SPLINE
SPL {X  -162.485, Y  +370.062, Z    +0.000, E1   +10.606, E3 +598080.502}
SPL {X  -162.818, Y  +379.636, Z    +0.000, E1    +5.115, E3 +598069.851}
SPL {X  -162.820, Y  +386.976, Z    +0.000, E1    +0.144, E3 +598068.950}
SPL {X  -162.820, Y  +391.982, Z    +0.000, E1    -3.443, E3 +598075.715}
SPL {X  -162.820, Y  +399.630, Z    +0.000, E1    -9.426, E3 +598078.222}
SPL {X  -162.820, Y  +408.127, Z    +0.000, E1   -18.417, E3 +598064.510}
SPL {X  -162.820, Y  +420.083, Z    +0.000, E1   -24.325, E3 +598084.986}
SPL {X  -162.820, Y  +428.527, Z    +0.000, E1   -26.988, E3 +598102.278}
SPL {X  -162.820, Y  +431.191, Z    +0.000, E1   -23.548, E3 +598137.131}
SPL {X  -162.820, Y  +432.946, Z    +0.000, E1   -22.795, E3 +598151.534}
SPL {X  -162.820, Y  +434.888, Z    +0.000, E1   -22.823, E3 +598160.941}
SPL {X  -162.820, Y  +436.834, Z    +0.000, E1   -22.779, E3 +598170.901}
SPL {X  -162.820, Y  +438.868, Z    +0.000, E1   -22.837, E3 +598180.555}
SPL {X  -162.820, Y  +441.351, Z    +0.000, E1   -22.805, E3 +598193.130}
SPL {X  -162.820, Y  +443.809, Z    +0.000, E1   -22.804, E3 +598205.296}
SPL {X  -162.820, Y  +446.105, Z    +0.000, E1   -22.815, E3 +598216.539}
SPL {X  -162.820, Y  +447.974, Z    +0.000, E1   -22.856, E3 +598225.441}
SPL {X  -162.820, Y  +449.911, Z    +0.000, E1   -22.774, E3 +598235.716}
SPL {X  -162.820, Y  +451.861, Z    +0.000, E1   -22.750, E3 +598245.564}
SPL {X  -162.820, Y  +454.167, Z    +0.000, E1   -22.842, E3 +598256.293}
SPL {X  -162.820, Y  +456.529, Z    +0.000, E1   -22.855, E3 +598267.822}
SPL {X  -162.820, Y  +458.725, Z    +0.000, E1   -22.793, E3 +598279.226}
SPL {X  -162.820, Y  +461.700, Z    +0.000, E1   -22.822, E3 +598293.849}
SPL {X  -162.820, Y  +464.633, Z    +0.000, E1   -22.813, E3 +598308.345}
SPL {X  -162.820, Y  +466.699, Z    +0.000, E1   -22.824, E3 +598318.391}
SPL {X  -162.820, Y  +468.655, Z    +0.000, E1   -22.858, E3 +598327.835}
SPL {X  -162.820, Y  +470.892, Z    +0.000, E1   -22.837, E3 +598339.074}
SPL {X  -162.820, Y  +473.485, Z    +0.000, E1   -22.806, E3 +598352.272}
SPL {X  -162.820, Y  +475.738, Z    +0.000, E1   -22.728, E3 +598363.937}
SPL {X  -162.820, Y  +478.177, Z    +0.000, E1   -22.834, E3 +598375.277}
SPL {X  -162.820, Y  +481.034, Z    +0.000, E1   -22.831, E3 +598389.414}
SPL {X  -162.820, Y  +483.391, Z    +0.000, E1   -22.793, E3 +598401.350}
SPL {X  -162.820, Y  +486.307, Z    +0.000, E1   -22.833, E3 +598415.604}
SPL {X  -162.820, Y  +489.750, Z    +0.000, E1   -22.832, E3 +598432.674}
SPL {X  -162.820, Y  +493.233, Z    +0.000, E1   -22.844, E3 +598449.811}
SPL {X  -162.820, Y  +496.150, Z    +0.000, E1   -22.796, E3 +598464.531}
SPL {X  -162.820, Y  +498.661, Z    +0.000, E1   -22.828, E3 +598476.712}
SPL {X  -162.820, Y  +501.761, Z    +0.000, E1   -22.820, E3 +598492.280}
SPL {X  -162.820, Y  +505.323, Z    +0.000, E1   -22.838, E3 +598509.727}
SPL {X  -162.820, Y  +507.875, Z    +0.000, E1   -22.849, E3 +598522.094}
SPL {X  -162.820, Y  +510.068, Z    +0.000, E1   -22.761, E3 +598533.787}
SPL {X  -162.820, Y  +512.359, Z    +0.000, E1   -22.823, E3 +598544.519}
SPL {X  -162.820, Y  +514.562, Z    +0.000, E1   -22.806, E3 +598555.706}
SPL {X  -162.820, Y  +517.952, Z    +0.000, E1   -22.864, E3 +598572.103}
SPL {X  -162.820, Y  +520.641, Z    +0.000, E1   -22.790, E3 +598585.821}
SPL {X  -162.820, Y  +522.740, Z    +0.000, E1   -22.811, E3 +598596.064}
SPL {X  -162.820, Y  +525.255, Z    +0.000, E1   -22.822, E3 +598608.484}
SPL {X  -162.820, Y  +528.050, Z    +0.000, E1   -22.808, E3 +598622.449}
SPL {X  -162.820, Y  +530.303, Z    +0.000, E1   -22.798, E3 +598633.603}
SPL {X  -162.820, Y  +532.614, Z    +0.000, E1   -22.828, E3 +598644.871}
SPL {X  -162.820, Y  +534.838, Z    +0.000, E1   -22.864, E3 +598655.500}
SPL {X  -162.820, Y  +536.882, Z    +0.000, E1   -22.782, E3 +598666.355}
SPL {X  -162.820, Y  +539.194, Z    +0.000, E1   -22.826, E3 +598677.404}
SPL {X  -162.820, Y  +541.555, Z    +0.000, E1   -22.817, E3 +598689.218}
SPL {X  -162.820, Y  +543.728, Z    +0.000, E1   -22.799, E3 +598700.076}
SPL {X  -162.820, Y  +545.925, Z    +0.000, E1   -22.803, E3 +598710.945}
SPL {X  -162.820, Y  +548.328, Z    +0.000, E1   -22.796, E3 +598722.941}
SPL {X  -162.820, Y  +551.027, Z    +0.000, E1   -22.819, E3 +598736.134}
SPL {X  -162.820, Y  +553.721, Z    +0.000, E1   -22.807, E3 +598749.578}
SPL {X  -162.820, Y  +556.430, Z    +0.000, E1   -22.821, E3 +598762.874}
SPL {X  -162.820, Y  +559.675, Z    +0.000, E1   -22.837, E3 +598778.954}
SPL {X  -162.820, Y  +562.799, Z    +0.000, E1   -22.814, E3 +598794.460}
SPL {X  -162.820, Y  +565.170, Z    +0.000, E1   -22.801, E3 +598806.285}
SPL {X  -162.820, Y  +568.020, Z    +0.000, E1   -22.787, E3 +598820.672}
SPL {X  -162.820, Y  +570.992, Z    +0.000, E1   -22.834, E3 +598834.891}
SPL {X  -162.820, Y  +573.634, Z    +0.000, E1   -22.827, E3 +598848.069}
SPL {X  -162.820, Y  +576.228, Z    +0.000, E1   -22.814, E3 +598860.965}
SPL {X  -162.820, Y  +578.553, Z    +0.000, E1   -22.801, E3 +598872.581}
SPL {X  -162.820, Y  +581.064, Z    +0.000, E1   -22.823, E3 +598884.866}
SPL {X  -162.820, Y  +583.435, Z    +0.000, E1   -22.808, E3 +598896.687}
SPL {X  -162.820, Y  +585.410, Z    +0.000, E1   -22.764, E3 +598906.823}
SPL {X  -162.820, Y  +587.676, Z    +0.000, E1   -22.853, E3 +598917.338}
SPL {X  -162.820, Y  +589.682, Z    +0.000, E1   -22.776, E3 +598927.868}
SPL {X  -162.820, Y  +591.720, Z    +0.000, E1   -22.868, E3 +598937.178}
SPL {X  -162.820, Y  +593.650, Z    +0.000, E1   -22.810, E3 +598947.248}
SPL {X  -162.820, Y  +595.830, Z    +0.000, E1   -22.828, E3 +598957.864}
SPL {X  -162.820, Y  +598.094, Z    +0.000, E1   -22.843, E3 +598968.977}
SPL {X  -162.820, Y  +600.420, Z    +0.000, E1   -22.826, E3 +598980.608}
SPL {X  -162.820, Y  +602.573, Z    +0.000, E1   -22.830, E3 +598991.194}
SPL {X  -162.820, Y  +604.828, Z    +0.000, E1   -22.784, E3 +599002.832}
SPL {X  -162.820, Y  +608.133, Z    +0.000, E1   -22.831, E3 +599018.950}
SPL {X  -162.820, Y  +611.103, Z    +0.000, E1   -22.785, E3 +599033.876}
SPL {X  -162.820, Y  +613.294, Z    +0.000, E1   -22.780, E3 +599044.749}
SPL {X  -162.820, Y  +615.356, Z    +0.000, E1   -22.799, E3 +599054.806}
SPL {X  -162.820, Y  +617.439, Z    +0.000, E1   -22.808, E3 +599065.064}
SPL {X  -162.820, Y  +619.665, Z    +0.000, E1   -22.817, E3 +599076.032}
SPL {X  -162.820, Y  +621.733, Z    +0.000, E1   -22.759, E3 +599086.756}
SPL {X  -162.820, Y  +624.076, Z    +0.000, E1   -22.774, E3 +599098.261}
SPL {X  -162.820, Y  +626.527, Z    +0.000, E1   -22.768, E3 +599110.504}
SPL {X  -162.820, Y  +629.758, Z    +0.000, E1   -22.800, E3 +599126.433}
SPL {X  -162.820, Y  +632.572, Z    +0.000, E1   -22.785, E3 +599140.282}
SPL {X  -162.820, Y  +634.507, Z    +0.000, E1   -22.784, E3 +599149.921}
SPL {X  -162.820, Y  +636.863, Z    +0.000, E1   -22.760, E3 +599161.843}
SPL {X  -162.820, Y  +640.111, Z    +0.000, E1   -22.809, E3 +599177.726}
SPL {X  -162.820, Y  +643.449, Z    +0.000, E1   -22.796, E3 +599194.244}
SPL {X  -162.820, Y  +645.630, Z    +0.000, E1   -22.795, E3 +599204.940}
SPL {X  -162.820, Y  +647.561, Z    +0.000, E1   -22.705, E3 +599215.390}
SPL {X  -162.820, Y  +649.758, Z    +0.000, E1   -22.780, E3 +599225.581}
SPL {X  -162.820, Y  +651.708, Z    +0.000, E1   -22.810, E3 +599235.075}
SPL {X  -162.820, Y  +653.898, Z    +0.000, E1   -22.796, E3 +599245.996}
SPL {X  -162.820, Y  +656.161, Z    +0.000, E1   -22.812, E3 +599257.117}
SPL {X  -162.820, Y  +658.384, Z    +0.000, E1   -22.822, E3 +599267.983}
SPL {X  -162.820, Y  +660.215, Z    +0.000, E1   -22.649, E3 +599278.574}
SPL {X  -162.820, Y  +662.823, Z    +0.000, E1   -22.799, E3 +599290.282}
SPL {X  -162.820, Y  +665.112, Z    +0.000, E1   -22.835, E3 +599301.336}
SPL {X  -162.820, Y  +667.016, Z    +0.000, E1   -22.823, E3 +599310.765}
SPL {X  -162.820, Y  +668.960, Z    +0.000, E1   -22.773, E3 +599320.932}
SPL {X  -162.820, Y  +672.333, Z    +0.000, E1   -22.837, E3 +599337.268}
SPL {X  -162.812, Y  +675.071, Z    +0.000, E1   -22.742, E3 +599351.413}
SPL {X  -162.773, Y  +677.428, Z    +0.000, E1   -22.762, E3 +599363.011}
SPL {X  -162.691, Y  +679.987, Z    +0.000, E1   -22.794, E3 +599375.424}
SPL {X  -162.604, Y  +681.880, Z    +0.000, E1   -22.691, E3 +599385.585}
SPL {X  -162.458, Y  +684.346, Z    +0.000, E1   -22.764, E3 +599397.379}
SPL {X  -162.296, Y  +686.547, Z    +0.000, E1   -22.660, E3 +599408.996}
SPL {X  -162.164, Y  +688.106, Z    +0.000, E1   -22.661, E3 +599416.729}
SPL {X  -161.938, Y  +690.422, Z    +0.000, E1   -22.769, E3 +599427.405}
SPL {X  -161.065, Y  +697.344, Z    +0.000, E1   -25.698, E3 +599436.524}
SPL {X  -158.730, Y  +709.763, Z    +0.000, E1   -31.225, E3 +599445.197}
ENDSPLINE

SPLINE
SPL {X  -160.932, Y  +698.225, Z    +0.000, E1   -21.712, E3 +599476.307}
SPL {X  -161.917, Y  +690.622, Z    +0.000, E1   -16.445, E3 +599489.907}
ENDSPLINE

SPLINE
SPL {X  -161.349, Y  +695.340, Z    +0.000, E1   -18.625, E3 +599497.526}
ENDSPLINE

SPLINE
SPL {X  -162.534, Y  +683.153, Z    +0.000, E1   -10.475, E3 +599518.657}
SPL {X  -162.820, Y  +667.630, Z    +0.000, E1    -0.882, E3 +599512.633}
SPL {X  -162.820, Y  +661.883, Z    +0.000, E1    +3.373, E3 +599518.076}
SPL {X  -162.820, Y  +655.163, Z    +0.000, E1    +8.702, E3 +599517.675}
SPL {X  -162.820, Y  +634.515, Z    +0.000, E1   +26.439, E3 +599510.088}
ENDSPLINE

SPLINE
SPL {X  -162.820, Y  +638.080, Z    +0.000, E1   +18.858, E3 +599540.053}
ENDSPLINE

SPLINE
SPL {X  -162.820, Y  +623.278, Z    +0.000, E1   +28.723, E3 +599541.623}
SPL {X  -162.820, Y  +618.658, Z    +0.000, E1   +26.841, E3 +599570.232}
ENDSPLINE

SPLINE
SPL {X  -162.820, Y  +623.685, Z    +0.000, E1   +22.346, E3 +599582.539}
ENDSPLINE

SPLINE
SPL {X  -162.820, Y  +621.304, Z    +0.000, E1   +22.259, E3 +599595.354}
SPL {X  -162.820, Y  +618.758, Z    +0.000, E1   +22.239, E3 +599608.505}
SPL {X  -162.820, Y  +616.062, Z    +0.000, E1   +22.275, E3 +599621.925}
SPL {X  -162.820, Y  +613.536, Z    +0.000, E1   +22.242, E3 +599635.047}
SPL {X  -162.820, Y  +610.461, Z    +0.000, E1   +22.264, E3 +599650.678}
SPL {X  -162.820, Y  +607.796, Z    +0.000, E1   +22.261, E3 +599664.049}
SPL {X  -162.820, Y  +605.178, Z    +0.000, E1   +22.267, E3 +599677.533}
SPL {X  -162.820, Y  +602.350, Z    +0.000, E1   +22.224, E3 +599692.150}
SPL {X  -162.820, Y  +599.842, Z    +0.000, E1   +22.298, E3 +599704.302}
SPL {X  -162.820, Y  +597.194, Z    +0.000, E1   +22.253, E3 +599718.223}
SPL {X  -162.820, Y  +594.115, Z    +0.000, E1   +22.273, E3 +599733.752}
SPL {X  -162.820, Y  +591.721, Z    +0.000, E1   +22.239, E3 +599746.067}
SPL {X  -162.820, Y  +589.492, Z    +0.000, E1   +22.304, E3 +599756.928}
SPL {X  -162.820, Y  +587.447, Z    +0.000, E1   +22.279, E3 +599767.457}
SPL {X  -162.820, Y  +585.192, Z    +0.000, E1   +22.298, E3 +599778.867}
SPL {X  -162.820, Y  +582.610, Z    +0.000, E1   +22.234, E3 +599792.490}
SPL {X  -162.820, Y  +580.317, Z    +0.000, E1   +22.300, E3 +599803.544}
SPL {X  -162.820, Y  +578.878, Z    +0.000, E1   +22.272, E3 +599811.054}
SPL {X  -162.820, Y  +576.856, Z    +0.000, E1   +22.233, E3 +599821.812}
SPL {X  -162.820, Y  +574.811, Z    +0.000, E1   +22.236, E3 +599832.076}
SPL {X  -162.820, Y  +572.645, Z    +0.000, E1   +22.246, E3 +599843.171}
SPL {X  -162.820, Y  +569.475, Z    +0.000, E1   +22.269, E3 +599859.177}
SPL {X  -162.820, Y  +565.838, Z    +0.000, E1   +22.271, E3 +599877.772}
SPL {X  -162.820, Y  +562.162, Z    +0.000, E1   +22.252, E3 +599896.589}
SPL {X  -162.820, Y  +559.515, Z    +0.000, E1   +22.273, E3 +599909.708}
SPL {X  -162.820, Y  +556.723, Z    +0.000, E1   +22.309, E3 +599923.792}
SPL {X  -162.820, Y  +553.294, Z    +0.000, E1   +22.266, E3 +599941.579}
SPL {X  -162.820, Y  +550.136, Z    +0.000, E1   +22.258, E3 +599957.693}
SPL {X  -162.820, Y  +546.694, Z    +0.000, E1   +22.290, E3 +599975.015}
SPL {X  -162.820, Y  +543.558, Z    +0.000, E1   +22.285, E3 +599990.878}
SPL {X  -162.820, Y  +541.633, Z    +0.000, E1   +22.257, E3 +600000.806}
SPL {X  -162.820, Y  +539.116, Z    +0.000, E1   +22.302, E3 +600013.416}
SPL {X  -162.820, Y  +536.913, Z    +0.000, E1   +22.192, E3 +600025.341}
SPL {X  -162.820, Y  +534.880, Z    +0.000, E1   +22.252, E3 +600035.294}
SPL {X  -162.820, Y  +532.896, Z    +0.000, E1   +22.234, E3 +600045.455}
SPL {X  -162.820, Y  +531.056, Z    +0.000, E1   +22.251, E3 +600054.737}
SPL {X  -162.820, Y  +528.708, Z    +0.000, E1   +22.319, E3 +600066.118}
SPL {X  -162.820, Y  +525.932, Z    +0.000, E1   +22.258, E3 +600080.875}
SPL {X  -162.820, Y  +522.524, Z    +0.000, E1   +22.326, E3 +600097.598}
SPL {X  -162.820, Y  +519.457, Z    +0.000, E1   +22.481, E3 +600111.727}
SPL {X  -162.820, Y  +506.285, Z    +0.000, E1   +28.538, E3 +600123.185}
SPL {X  -162.820, Y  +504.441, Z    +0.000, E1   +27.574, E3 +600137.528}
SPL {X  -162.820, Y  +502.813, Z    +0.000, E1   +26.013, E3 +600155.725}
SPL {X  -162.820, Y  +502.016, Z    +0.000, E1   +24.802, E3 +600168.068}
SPL {X  -162.820, Y  +501.060, Z    +0.000, E1   +24.081, E3 +600178.257}
SPL {X  -162.820, Y  +499.934, Z    +0.000, E1   +22.814, E3 +600194.126}
SPL {X  -162.820, Y  +498.303, Z    +0.000, E1   +21.749, E3 +600211.382}
SPL {X  -162.820, Y  +495.897, Z    +0.000, E1   +21.662, E3 +600224.536}
SPL {X  -162.820, Y  +493.717, Z    +0.000, E1   +21.704, E3 +600235.642}
SPL {X  -162.820, Y  +491.396, Z    +0.000, E1   +21.707, E3 +600247.766}
SPL {X  -162.820, Y  +489.485, Z    +0.000, E1   +21.661, E3 +600258.114}
SPL {X  -162.820, Y  +487.723, Z    +0.000, E1   +21.665, E3 +600267.317}
SPL {X  -162.820, Y  +485.661, Z    +0.000, E1   +21.712, E3 +600277.761}
SPL {X  -162.820, Y  +482.775, Z    +0.000, E1   +21.716, E3 +600293.013}
SPL {X  -162.820, Y  +479.894, Z    +0.000, E1   +21.695, E3 +600308.089}
SPL {X  -162.820, Y  +477.685, Z    +0.000, E1   +21.656, E3 +600320.027}
SPL {X  -162.820, Y  +475.419, Z    +0.000, E1   +21.711, E3 +600331.380}
SPL {X  -162.820, Y  +473.301, Z    +0.000, E1   +21.712, E3 +600342.477}
SPL {X  -162.820, Y  +470.965, Z    +0.000, E1   +21.700, E3 +600354.822}
SPL {X  -162.820, Y  +469.036, Z    +0.000, E1   +21.695, E3 +600364.865}
SPL {X  -162.820, Y  +467.138, Z    +0.000, E1   +21.678, E3 +600375.037}
SPL {X  -162.820, Y  +465.011, Z    +0.000, E1   +21.692, E3 +600386.020}
SPL {X  -162.820, Y  +462.669, Z    +0.000, E1   +21.752, E3 +600397.800}
SPL {X  -162.820, Y  +460.725, Z    +0.000, E1   +21.689, E3 +600408.413}
SPL {X  -162.820, Y  +458.666, Z    +0.000, E1   +21.695, E3 +600419.225}
SPL {X  -162.820, Y  +456.431, Z    +0.000, E1   +21.708, E3 +600430.753}
SPL {X  -162.820, Y  +454.628, Z    +0.000, E1   +21.674, E3 +600440.472}
SPL {X  -162.820, Y  +452.690, Z    +0.000, E1   +21.773, E3 +600449.746}
SPL {X  -162.820, Y  +450.610, Z    +0.000, E1   +21.698, E3 +600461.345}
SPL {X  -162.820, Y  +448.170, Z    +0.000, E1   +21.667, E3 +600474.365}
SPL {X  -162.820, Y  +446.246, Z    +0.000, E1   +21.696, E3 +600484.183}
SPL {X  -162.820, Y  +443.784, Z    +0.000, E1   +21.713, E3 +600496.969}
SPL {X  -162.820, Y  +440.567, Z    +0.000, E1   +21.731, E3 +600513.809}
SPL {X  -162.820, Y  +437.628, Z    +0.000, E1   +21.678, E3 +600529.473}
SPL {X  -162.820, Y  +435.262, Z    +0.000, E1   +21.727, E3 +600541.409}
SPL {X  -162.820, Y  +433.510, Z    +0.000, E1   +21.692, E3 +600550.823}
SPL {X  -162.820, Y  +431.492, Z    +0.000, E1   +21.686, E3 +600561.518}
SPL {X  -162.820, Y  +429.074, Z    +0.000, E1   +21.710, E3 +600573.970}
SPL {X  -162.820, Y  +427.020, Z    +0.000, E1   +21.674, E3 +600584.972}
SPL {X  -162.820, Y  +424.525, Z    +0.000, E1   +21.712, E3 +600597.885}
SPL {X  -162.820, Y  +421.144, Z    +0.000, E1   +21.719, E3 +600615.552}
SPL {X  -162.820, Y  +418.116, Z    +0.000, E1   +21.761, E3 +600630.883}
SPL {X  -162.820, Y  +416.127, Z    +0.000, E1   +21.715, E3 +600641.588}
SPL {X  -162.820, Y  +414.361, Z    +0.000, E1   +21.613, E3 +600651.775}
SPL {X  -162.820, Y  +412.134, Z    +0.000, E1   +21.697, E3 +600662.720}
SPL {X  -162.820, Y  +409.248, Z    +0.000, E1   +21.741, E3 +600677.655}
SPL {X  -162.820, Y  +406.238, Z    +0.000, E1   +21.697, E3 +600693.623}
SPL {X  -162.820, Y  +404.001, Z    +0.000, E1   +21.723, E3 +600705.053}
SPL {X  -162.820, Y  +402.223, Z    +0.000, E1   +21.697, E3 +600714.538}
SPL {X  -162.820, Y  +400.348, Z    +0.000, E1   +21.713, E3 +600724.264}
SPL {X  -162.820, Y  +398.298, Z    +0.000, E1   +21.721, E3 +600734.879}
SPL {X  -162.820, Y  +396.371, Z    +0.000, E1   +21.713, E3 +600745.061}
SPL {X  -162.820, Y  +394.508, Z    +0.000, E1   +21.616, E3 +600755.617}
SPL {X  -162.820, Y  +392.435, Z    +0.000, E1   +21.681, E3 +600765.970}
SPL {X  -162.820, Y  +389.390, Z    +0.000, E1   +21.742, E3 +600781.577}
SPL {X  -162.820, Y  +386.818, Z    +0.000, E1   +21.679, E3 +600795.336}
SPL {X  -162.820, Y  +384.697, Z    +0.000, E1   +21.693, E3 +600806.406}
SPL {X  -162.820, Y  +382.288, Z    +0.000, E1   +21.742, E3 +600818.529}
SPL {X  -162.817, Y  +379.520, Z    +0.000, E1   +21.723, E3 +600833.367}
SPL {X  -162.776, Y  +376.710, Z    +0.000, E1   +21.698, E3 +600848.106}
SPL {X  -162.707, Y  +374.438, Z    +0.000, E1   +21.688, E3 +600860.110}
SPL {X  -162.607, Y  +372.171, Z    +0.000, E1   +21.692, E3 +600871.910}
SPL {X  -162.494, Y  +370.197, Z    +0.000, E1   +21.655, E3 +600882.536}
SPL {X  -162.349, Y  +368.131, Z    +0.000, E1   +21.624, E3 +600893.654}
SPL {X  -162.161, Y  +365.866, Z    +0.000, E1   +21.642, E3 +600905.339}
SPL {X  -161.651, Y  +361.024, Z    +0.000, E1   +22.970, E3 +600918.762}
SPL {X  -160.281, Y  +351.857, Z    +0.000, E1   +24.243, E3 +600954.101}
ENDSPLINE

SPLINE
SPL {X  -161.833, Y  +362.603, Z    +0.000, E1   +17.021, E3 +600968.797}
ENDSPLINE

SPLINE
SPL {X  -160.786, Y  +354.842, Z    +0.000, E1   +19.274, E3 +601000.953}
ENDSPLINE

SPLINE
SPL {X  -162.485, Y  +370.062, Z    +0.000, E1   +10.606, E3 +601007.331}
SPL {X  -162.818, Y  +379.636, Z    +0.000, E1    +5.115, E3 +600996.680}
SPL {X  -162.820, Y  +386.976, Z    +0.000, E1    +0.144, E3 +600995.779}
SPL {X  -162.820, Y  +391.982, Z    +0.000, E1    -3.443, E3 +601002.544}
SPL {X  -162.820, Y  +399.630, Z    +0.000, E1    -9.426, E3 +601005.051}
SPL {X  -162.820, Y  +408.127, Z    +0.000, E1   -18.417, E3 +600991.340}
SPL {X  -162.820, Y  +420.083, Z    +0.000, E1   -24.325, E3 +601011.815}
SPL {X  -162.820, Y  +428.527, Z    +0.000, E1   -26.988, E3 +601029.107}
SPL {X  -162.820, Y  +431.336, Z    +0.000, E1   -24.162, E3 +601059.317}
SPL {X  -162.820, Y  +432.048, Z    +0.000, E1   -22.832, E3 +601073.821}
SPL {X  -162.820, Y  +434.888, Z    +0.000, E1   -22.823, E3 +601087.770}
SPL {X  -162.820, Y  +436.834, Z    +0.000, E1   -22.779, E3 +601097.730}
SPL {X  -162.820, Y  +438.868, Z    +0.000, E1   -22.837, E3 +601107.384}
SPL {X  -162.820, Y  +441.351, Z    +0.000, E1   -22.805, E3 +601119.959}
SPL {X  -162.820, Y  +443.809, Z    +0.000, E1   -22.804, E3 +601132.126}
SPL {X  -162.820, Y  +446.105, Z    +0.000, E1   -22.815, E3 +601143.368}
SPL {X  -162.820, Y  +447.974, Z    +0.000, E1   -22.856, E3 +601152.271}
SPL {X  -162.820, Y  +449.911, Z    +0.000, E1   -22.774, E3 +601162.546}
SPL {X  -162.820, Y  +451.861, Z    +0.000, E1   -22.750, E3 +601172.393}
SPL {X  -162.820, Y  +454.167, Z    +0.000, E1   -22.842, E3 +601183.123}
SPL {X  -162.820, Y  +456.529, Z    +0.000, E1   -22.855, E3 +601194.651}
SPL {X  -162.820, Y  +458.725, Z    +0.000, E1   -22.793, E3 +601206.055}
SPL {X  -162.820, Y  +460.754, Z    +0.000, E1   -22.806, E3 +601215.928}
SPL {X  -162.820, Y  +462.409, Z    +0.000, E1   -22.783, E3 +601224.345}
SPL {X  -162.820, Y  +464.633, Z    +0.000, E1   -22.813, E3 +601235.175}
SPL {X  -162.820, Y  +467.913, Z    +0.000, E1   -22.879, E3 +601251.014}
SPL {X  -162.820, Y  +470.892, Z    +0.000, E1   -22.837, E3 +601265.903}
SPL {X  -162.820, Y  +472.726, Z    +0.000, E1   -22.777, E3 +601275.442}
SPL {X  -162.820, Y  +475.118, Z    +0.000, E1   -22.777, E3 +601287.413}
SPL {X  -162.820, Y  +477.389, Z    +0.000, E1   -22.803, E3 +601298.330}
SPL {X  -162.820, Y  +478.914, Z    +0.000, E1   -22.821, E3 +601305.721}
SPL {X  -162.820, Y  +481.034, Z    +0.000, E1   -22.831, E3 +601316.244}
SPL {X  -162.820, Y  +484.256, Z    +0.000, E1   -22.840, E3 +601332.262}
SPL {X  -162.820, Y  +487.952, Z    +0.000, E1   -22.824, E3 +601350.692}
SPL {X  -162.820, Y  +490.653, Z    +0.000, E1   -22.810, E3 +601363.962}
SPL {X  -162.820, Y  +493.233, Z    +0.000, E1   -22.844, E3 +601376.640}
SPL {X  -162.820, Y  +496.150, Z    +0.000, E1   -22.796, E3 +601391.360}
SPL {X  -162.820, Y  +498.661, Z    +0.000, E1   -22.828, E3 +601403.541}
SPL {X  -162.820, Y  +501.761, Z    +0.000, E1   -22.820, E3 +601419.109}
SPL {X  -162.820, Y  +505.323, Z    +0.000, E1   -22.838, E3 +601436.556}
SPL {X  -162.820, Y  +507.875, Z    +0.000, E1   -22.849, E3 +601448.923}
SPL {X  -162.820, Y  +510.068, Z    +0.000, E1   -22.761, E3 +601460.616}
SPL {X  -162.820, Y  +512.359, Z    +0.000, E1   -22.823, E3 +601471.348}
SPL {X  -162.820, Y  +514.562, Z    +0.000, E1   -22.806, E3 +601482.535}
SPL {X  -162.820, Y  +517.952, Z    +0.000, E1   -22.864, E3 +601498.932}
SPL {X  -162.820, Y  +520.641, Z    +0.000, E1   -22.790, E3 +601512.651}
SPL {X  -162.820, Y  +522.740, Z    +0.000, E1   -22.811, E3 +601522.893}
SPL {X  -162.820, Y  +524.628, Z    +0.000, E1   -22.846, E3 +601531.888}
SPL {X  -162.820, Y  +526.661, Z    +0.000, E1   -22.801, E3 +601542.444}
SPL {X  -162.820, Y  +529.662, Z    +0.000, E1   -22.810, E3 +601557.294}
SPL {X  -162.820, Y  +532.614, Z    +0.000, E1   -22.828, E3 +601571.701}
SPL {X  -162.820, Y  +534.838, Z    +0.000, E1   -22.864, E3 +601582.330}
SPL {X  -162.820, Y  +536.882, Z    +0.000, E1   -22.782, E3 +601593.184}
SPL {X  -162.820, Y  +539.194, Z    +0.000, E1   -22.826, E3 +601604.233}
SPL {X  -162.820, Y  +541.555, Z    +0.000, E1   -22.817, E3 +601616.047}
SPL {X  -162.820, Y  +543.728, Z    +0.000, E1   -22.799, E3 +601626.905}
SPL {X  -162.820, Y  +545.925, Z    +0.000, E1   -22.803, E3 +601637.775}
SPL {X  -162.820, Y  +548.328, Z    +0.000, E1   -22.796, E3 +601649.770}
SPL {X  -162.820, Y  +551.027, Z    +0.000, E1   -22.819, E3 +601662.963}
SPL {X  -162.820, Y  +553.721, Z    +0.000, E1   -22.807, E3 +601676.407}
SPL {X  -162.820, Y  +556.430, Z    +0.000, E1   -22.821, E3 +601689.703}
SPL {X  -162.820, Y  +558.974, Z    +0.000, E1   -22.806, E3 +601702.403}
SPL {X  -162.820, Y  +562.171, Z    +0.000, E1   -22.845, E3 +601718.101}
SPL {X  -162.820, Y  +565.170, Z    +0.000, E1   -22.801, E3 +601733.115}
SPL {X  -162.820, Y  +567.308, Z    +0.000, E1   -22.750, E3 +601744.131}
SPL {X  -162.820, Y  +570.378, Z    +0.000, E1   -22.843, E3 +601758.755}
SPL {X  -162.820, Y  +573.634, Z    +0.000, E1   -22.827, E3 +601774.898}
SPL {X  -162.820, Y  +576.228, Z    +0.000, E1   -22.814, E3 +601787.795}
SPL {X  -162.820, Y  +578.553, Z    +0.000, E1   -22.801, E3 +601799.411}
SPL {X  -162.820, Y  +581.064, Z    +0.000, E1   -22.823, E3 +601811.695}
SPL {X  -162.820, Y  +583.435, Z    +0.000, E1   -22.808, E3 +601823.517}
SPL {X  -162.820, Y  +585.410, Z    +0.000, E1   -22.764, E3 +601833.652}
SPL {X  -162.820, Y  +587.676, Z    +0.000, E1   -22.853, E3 +601844.167}
SPL {X  -162.820, Y  +590.707, Z    +0.000, E1   -22.855, E3 +601859.317}
SPL {X  -162.820, Y  +593.650, Z    +0.000, E1   -22.810, E3 +601874.078}
SPL {X  -162.820, Y  +595.830, Z    +0.000, E1   -22.828, E3 +601884.693}
SPL {X  -162.820, Y  +598.094, Z    +0.000, E1   -22.843, E3 +601895.807}
SPL {X  -162.820, Y  +600.420, Z    +0.000, E1   -22.826, E3 +601907.438}
SPL {X  -162.820, Y  +602.573, Z    +0.000, E1   -22.830, E3 +601918.023}
SPL {X  -162.820, Y  +604.828, Z    +0.000, E1   -22.784, E3 +601929.661}
SPL {X  -162.820, Y  +608.133, Z    +0.000, E1   -22.831, E3 +601945.779}
SPL {X  -162.820, Y  +611.103, Z    +0.000, E1   -22.785, E3 +601960.705}
SPL {X  -162.820, Y  +613.294, Z    +0.000, E1   -22.780, E3 +601971.578}
SPL {X  -162.820, Y  +615.356, Z    +0.000, E1   -22.799, E3 +601981.635}
SPL {X  -162.820, Y  +617.439, Z    +0.000, E1   -22.808, E3 +601991.893}
SPL {X  -162.820, Y  +619.665, Z    +0.000, E1   -22.817, E3 +602002.861}
SPL {X  -162.820, Y  +621.733, Z    +0.000, E1   -22.759, E3 +602013.586}
SPL {X  -162.820, Y  +624.076, Z    +0.000, E1   -22.774, E3 +602025.091}
SPL {X  -162.820, Y  +627.244, Z    +0.000, E1   -22.803, E3 +602040.773}
SPL {X  -162.820, Y  +630.349, Z    +0.000, E1   -22.766, E3 +602056.305}
SPL {X  -162.820, Y  +632.572, Z    +0.000, E1   -22.785, E3 +602067.111}
SPL {X  -162.820, Y  +634.507, Z    +0.000, E1   -22.784, E3 +602076.750}
SPL {X  -162.820, Y  +636.863, Z    +0.000, E1   -22.760, E3 +602088.672}
SPL {X  -162.820, Y  +640.111, Z    +0.000, E1   -22.809, E3 +602104.555}
SPL {X  -162.820, Y  +643.449, Z    +0.000, E1   -22.796, E3 +602121.073}
SPL {X  -162.820, Y  +645.630, Z    +0.000, E1   -22.795, E3 +602131.769}
SPL {X  -162.820, Y  +647.561, Z    +0.000, E1   -22.705, E3 +602142.220}
SPL {X  -162.820, Y  +651.051, Z    +0.000, E1   -22.833, E3 +602158.639}
SPL {X  -162.820, Y  +653.898, Z    +0.000, E1   -22.796, E3 +602172.825}
SPL {X  -162.820, Y  +656.161, Z    +0.000, E1   -22.812, E3 +602183.946}
SPL {X  -162.820, Y  +658.384, Z    +0.000, E1   -22.822, E3 +602194.813}
SPL {X  -162.820, Y  +660.215, Z    +0.000, E1   -22.649, E3 +602205.403}
SPL {X  -162.820, Y  +662.823, Z    +0.000, E1   -22.799, E3 +602217.111}
SPL {X  -162.820, Y  +665.112, Z    +0.000, E1   -22.835, E3 +602228.166}
SPL {X  -162.820, Y  +667.016, Z    +0.000, E1   -22.823, E3 +602237.594}
SPL {X  -162.820, Y  +668.960, Z    +0.000, E1   -22.773, E3 +602247.762}
SPL {X  -162.820, Y  +672.333, Z    +0.000, E1   -22.837, E3 +602264.098}
SPL {X  -162.812, Y  +675.071, Z    +0.000, E1   -22.742, E3 +602278.243}
SPL {X  -162.773, Y  +677.428, Z    +0.000, E1   -22.762, E3 +602289.840}
SPL {X  -162.691, Y  +679.987, Z    +0.000, E1   -22.794, E3 +602302.254}
SPL {X  -162.559, Y  +682.717, Z    +0.000, E1   -22.726, E3 +602316.437}
SPL {X  -162.349, Y  +685.880, Z    +0.000, E1   -22.738, E3 +602332.038}
SPL {X  -162.164, Y  +688.106, Z    +0.000, E1   -22.661, E3 +602343.558}
SPL {X  -161.938, Y  +690.422, Z    +0.000, E1   -22.769, E3 +602354.234}
SPL {X  -161.065, Y  +697.344, Z    +0.000, E1   -25.698, E3 +602363.353}
SPL {X  -158.553, Y  +710.529, Z    +0.000, E1   -30.890, E3 +602377.250}
ENDSPLINE

SPLINE
SPL {X  -161.215, Y  +696.305, Z    +0.000, E1   -20.575, E3 +602403.831}
SPL {X  -161.691, Y  +692.643, Z    +0.000, E1   -17.369, E3 +602420.019}
SPL {X  -162.534, Y  +683.153, Z    +0.000, E1   -10.475, E3 +602445.486}
SPL {X  -162.820, Y  +667.630, Z    +0.000, E1    -0.882, E3 +602439.462}
SPL {X  -162.820, Y  +661.883, Z    +0.000, E1    +3.373, E3 +602444.905}
SPL {X  -162.820, Y  +655.163, Z    +0.000, E1    +8.702, E3 +602444.504}
SPL {X  -162.820, Y  +634.515, Z    +0.000, E1   +26.439, E3 +602436.917}
ENDSPLINE

SPLINE
SPL {X  -162.820, Y  +638.080, Z    +0.000, E1   +18.858, E3 +602466.882}
ENDSPLINE

SPLINE
SPL {X  -162.820, Y  +623.278, Z    +0.000, E1   +28.723, E3 +602468.453}
SPL {X  -162.820, Y  +611.829, Z    +0.000, E1   +31.229, E3 +602492.105}
ENDSPLINE

SPLINE
SPL {X  -162.820, Y  +623.595, Z    +0.000, E1   +22.712, E3 +602507.026}
ENDSPLINE

SPLINE
SPL {X  -162.820, Y  +621.304, Z    +0.000, E1   +22.259, E3 +602522.183}
SPL {X  -162.820, Y  +618.758, Z    +0.000, E1   +22.239, E3 +602535.334}
SPL {X  -162.820, Y  +616.062, Z    +0.000, E1   +22.275, E3 +602548.755}
SPL {X  -162.820, Y  +613.536, Z    +0.000, E1   +22.242, E3 +602561.876}
SPL {X  -162.820, Y  +611.128, Z    +0.000, E1   +22.252, E3 +602574.047}
SPL {X  -162.820, Y  +608.428, Z    +0.000, E1   +22.255, E3 +602587.830}
SPL {X  -162.820, Y  +605.984, Z    +0.000, E1   +22.221, E3 +602600.467}
SPL {X  -162.820, Y  +603.020, Z    +0.000, E1   +22.272, E3 +602615.366}
SPL {X  -162.820, Y  +599.168, Z    +0.000, E1   +22.310, E3 +602634.633}
SPL {X  -162.820, Y  +596.569, Z    +0.000, E1   +22.222, E3 +602648.356}
SPL {X  -162.820, Y  +594.115, Z    +0.000, E1   +22.273, E3 +602660.581}
SPL {X  -162.820, Y  +591.721, Z    +0.000, E1   +22.239, E3 +602672.896}
SPL {X  -162.820, Y  +589.492, Z    +0.000, E1   +22.304, E3 +602683.757}
SPL {X  -162.820, Y  +586.660, Z    +0.000, E1   +22.307, E3 +602698.198}
SPL {X  -162.820, Y  +583.204, Z    +0.000, E1   +22.278, E3 +602716.103}
SPL {X  -162.820, Y  +580.317, Z    +0.000, E1   +22.300, E3 +602730.373}
SPL {X  -162.820, Y  +578.061, Z    +0.000, E1   +22.264, E3 +602742.258}
SPL {X  -162.820, Y  +575.394, Z    +0.000, E1   +22.240, E3 +602756.003}
SPL {X  -162.820, Y  +573.156, Z    +0.000, E1   +22.254, E3 +602767.213}
SPL {X  -162.820, Y  +570.852, Z    +0.000, E1   +22.234, E3 +602779.237}
SPL {X  -162.820, Y  +568.608, Z    +0.000, E1   +22.253, E3 +602790.370}
SPL {X  -162.820, Y  +565.838, Z    +0.000, E1   +22.271, E3 +602804.601}
SPL {X  -162.820, Y  +562.162, Z    +0.000, E1   +22.252, E3 +602823.418}
SPL {X  -162.820, Y  +558.919, Z    +0.000, E1   +22.286, E3 +602839.582}
SPL {X  -162.820, Y  +556.169, Z    +0.000, E1   +22.295, E3 +602853.411}
SPL {X  -162.820, Y  +553.294, Z    +0.000, E1   +22.266, E3 +602868.409}
SPL {X  -162.820, Y  +550.136, Z    +0.000, E1   +22.258, E3 +602884.522}
SPL {X  -162.820, Y  +546.694, Z    +0.000, E1   +22.290, E3 +602901.844}
SPL {X  -162.820, Y  +543.558, Z    +0.000, E1   +22.285, E3 +602917.707}
SPL {X  -162.820, Y  +541.633, Z    +0.000, E1   +22.257, E3 +602927.635}
SPL {X  -162.820, Y  +539.116, Z    +0.000, E1   +22.302, E3 +602940.246}
SPL {X  -162.820, Y  +536.913, Z    +0.000, E1   +22.192, E3 +602952.170}
SPL {X  -162.820, Y  +534.880, Z    +0.000, E1   +22.252, E3 +602962.124}
SPL {X  -162.820, Y  +532.896, Z    +0.000, E1   +22.234, E3 +602972.284}
SPL {X  -162.820, Y  +531.056, Z    +0.000, E1   +22.251, E3 +602981.566}
SPL {X  -162.820, Y  +528.708, Z    +0.000, E1   +22.319, E3 +602992.948}
SPL {X  -162.820, Y  +525.932, Z    +0.000, E1   +22.258, E3 +603007.704}
SPL {X  -162.820, Y  +522.524, Z    +0.000, E1   +22.326, E3 +603024.428}
SPL {X  -162.820, Y  +519.457, Z    +0.000, E1   +22.481, E3 +603038.557}
SPL {X  -162.820, Y  +506.285, Z    +0.000, E1   +28.538, E3 +603050.015}
SPL {X  -162.820, Y  +504.441, Z    +0.000, E1   +27.574, E3 +603064.357}
SPL {X  -162.820, Y  +502.813, Z    +0.000, E1   +26.013, E3 +603082.554}
SPL {X  -162.820, Y  +502.016, Z    +0.000, E1   +24.802, E3 +603094.897}
SPL {X  -162.820, Y  +501.060, Z    +0.000, E1   +24.081, E3 +603105.086}
SPL {X  -162.820, Y  +499.934, Z    +0.000, E1   +22.814, E3 +603120.955}
SPL {X  -162.820, Y  +498.303, Z    +0.000, E1   +21.749, E3 +603138.211}
SPL {X  -162.820, Y  +495.897, Z    +0.000, E1   +21.662, E3 +603151.365}
SPL {X  -162.820, Y  +493.717, Z    +0.000, E1   +21.704, E3 +603162.471}
SPL {X  -162.820, Y  +491.396, Z    +0.000, E1   +21.707, E3 +603174.595}
SPL {X  -162.820, Y  +489.485, Z    +0.000, E1   +21.661, E3 +603184.943}
SPL {X  -162.820, Y  +487.723, Z    +0.000, E1   +21.665, E3 +603194.146}
SPL {X  -162.820, Y  +485.661, Z    +0.000, E1   +21.712, E3 +603204.590}
SPL {X  -162.820, Y  +482.775, Z    +0.000, E1   +21.716, E3 +603219.842}
SPL {X  -162.820, Y  +479.894, Z    +0.000, E1   +21.695, E3 +603234.919}
SPL {X  -162.820, Y  +477.685, Z    +0.000, E1   +21.656, E3 +603246.856}
SPL {X  -162.820, Y  +475.419, Z    +0.000, E1   +21.711, E3 +603258.209}
SPL {X  -162.820, Y  +473.301, Z    +0.000, E1   +21.712, E3 +603269.306}
SPL {X  -162.820, Y  +470.965, Z    +0.000, E1   +21.700, E3 +603281.651}
SPL {X  -162.820, Y  +469.036, Z    +0.000, E1   +21.695, E3 +603291.695}
SPL {X  -162.820, Y  +467.138, Z    +0.000, E1   +21.678, E3 +603301.866}
SPL {X  -162.820, Y  +465.011, Z    +0.000, E1   +21.692, E3 +603312.849}
SPL {X  -162.820, Y  +462.669, Z    +0.000, E1   +21.752, E3 +603324.629}
SPL {X  -162.820, Y  +460.725, Z    +0.000, E1   +21.689, E3 +603335.242}
SPL {X  -162.820, Y  +458.666, Z    +0.000, E1   +21.695, E3 +603346.054}
SPL {X  -162.820, Y  +456.431, Z    +0.000, E1   +21.708, E3 +603357.583}
SPL {X  -162.820, Y  +454.628, Z    +0.000, E1   +21.674, E3 +603367.301}
SPL {X  -162.820, Y  +452.690, Z    +0.000, E1   +21.773, E3 +603376.575}
SPL {X  -162.820, Y  +450.610, Z    +0.000, E1   +21.698, E3 +603388.174}
SPL {X  -162.820, Y  +448.170, Z    +0.000, E1   +21.667, E3 +603401.195}
SPL {X  -162.820, Y  +446.246, Z    +0.000, E1   +21.696, E3 +603411.012}
SPL {X  -162.820, Y  +443.784, Z    +0.000, E1   +21.713, E3 +603423.799}
SPL {X  -162.820, Y  +440.567, Z    +0.000, E1   +21.731, E3 +603440.638}
SPL {X  -162.820, Y  +437.628, Z    +0.000, E1   +21.678, E3 +603456.303}
SPL {X  -162.820, Y  +435.262, Z    +0.000, E1   +21.727, E3 +603468.238}
SPL {X  -162.820, Y  +433.510, Z    +0.000, E1   +21.692, E3 +603477.652}
SPL {X  -162.820, Y  +431.492, Z    +0.000, E1   +21.686, E3 +603488.347}
SPL {X  -162.820, Y  +429.074, Z    +0.000, E1   +21.710, E3 +603500.799}
SPL {X  -162.820, Y  +427.020, Z    +0.000, E1   +21.674, E3 +603511.801}
SPL {X  -162.820, Y  +424.525, Z    +0.000, E1   +21.712, E3 +603524.714}
SPL {X  -162.820, Y  +421.144, Z    +0.000, E1   +21.719, E3 +603542.381}
SPL {X  -162.820, Y  +418.116, Z    +0.000, E1   +21.761, E3 +603557.712}
SPL {X  -162.820, Y  +416.127, Z    +0.000, E1   +21.715, E3 +603568.417}
SPL {X  -162.820, Y  +414.361, Z    +0.000, E1   +21.613, E3 +603578.604}
SPL {X  -162.820, Y  +412.134, Z    +0.000, E1   +21.697, E3 +603589.549}
SPL {X  -162.820, Y  +409.248, Z    +0.000, E1   +21.741, E3 +603604.484}
SPL {X  -162.820, Y  +406.238, Z    +0.000, E1   +21.697, E3 +603620.452}
SPL {X  -162.820, Y  +404.001, Z    +0.000, E1   +21.723, E3 +603631.882}
SPL {X  -162.820, Y  +402.223, Z    +0.000, E1   +21.697, E3 +603641.367}
SPL {X  -162.820, Y  +400.348, Z    +0.000, E1   +21.713, E3 +603651.093}
SPL {X  -162.820, Y  +398.298, Z    +0.000, E1   +21.721, E3 +603661.709}
SPL {X  -162.820, Y  +396.371, Z    +0.000, E1   +21.713, E3 +603671.890}
SPL {X  -162.820, Y  +394.508, Z    +0.000, E1   +21.616, E3 +603682.446}
SPL {X  -162.820, Y  +392.435, Z    +0.000, E1   +21.681, E3 +603692.799}
SPL {X  -162.820, Y  +389.390, Z    +0.000, E1   +21.742, E3 +603708.406}
SPL {X  -162.820, Y  +386.818, Z    +0.000, E1   +21.679, E3 +603722.165}
SPL {X  -162.820, Y  +384.697, Z    +0.000, E1   +21.693, E3 +603733.235}
SPL {X  -162.820, Y  +382.288, Z    +0.000, E1   +21.742, E3 +603745.359}
SPL {X  -162.817, Y  +379.520, Z    +0.000, E1   +21.723, E3 +603760.196}
SPL {X  -162.776, Y  +376.710, Z    +0.000, E1   +21.698, E3 +603774.935}
SPL {X  -162.707, Y  +374.438, Z    +0.000, E1   +21.688, E3 +603786.939}
SPL {X  -162.607, Y  +372.171, Z    +0.000, E1   +21.692, E3 +603798.739}
SPL {X  -162.494, Y  +370.197, Z    +0.000, E1   +21.655, E3 +603809.365}
SPL {X  -162.349, Y  +368.131, Z    +0.000, E1   +21.624, E3 +603820.483}
SPL {X  -162.161, Y  +365.866, Z    +0.000, E1   +21.642, E3 +603832.168}
SPL {X  -161.651, Y  +361.024, Z    +0.000, E1   +22.970, E3 +603845.592}
SPL {X  -160.281, Y  +351.857, Z    +0.000, E1   +24.243, E3 +603880.931}
ENDSPLINE

SPLINE
SPL {X  -161.833, Y  +362.603, Z    +0.000, E1   +17.021, E3 +603895.627}
ENDSPLINE

SPLINE
SPL {X  -160.786, Y  +354.842, Z    +0.000, E1   +19.274, E3 +603927.782}
ENDSPLINE

SPLINE
SPL {X  -162.485, Y  +370.062, Z    +0.000, E1   +10.606, E3 +603934.160}
SPL {X  -162.818, Y  +379.636, Z    +0.000, E1    +5.115, E3 +603923.509}
SPL {X  -162.820, Y  +386.976, Z    +0.000, E1    +0.144, E3 +603922.608}
SPL {X  -162.820, Y  +391.982, Z    +0.000, E1    -3.443, E3 +603929.373}
SPL {X  -162.820, Y  +399.630, Z    +0.000, E1    -9.426, E3 +603931.880}
SPL {X  -162.820, Y  +408.127, Z    +0.000, E1   -18.417, E3 +603918.169}
SPL {X  -162.820, Y  +420.083, Z    +0.000, E1   -24.325, E3 +603938.644}
SPL {X  -162.820, Y  +428.527, Z    +0.000, E1   -26.988, E3 +603955.936}
SPL {X  -162.820, Y  +431.336, Z    +0.000, E1   -24.162, E3 +603986.146}
SPL {X  -162.820, Y  +432.048, Z    +0.000, E1   -22.832, E3 +604000.650}
SPL {X  -162.820, Y  +434.888, Z    +0.000, E1   -22.823, E3 +604014.600}
SPL {X  -162.820, Y  +436.834, Z    +0.000, E1   -22.779, E3 +604024.560}
SPL {X  -162.820, Y  +438.868, Z    +0.000, E1   -22.837, E3 +604034.213}
SPL {X  -162.820, Y  +441.351, Z    +0.000, E1   -22.805, E3 +604046.789}
SPL {X  -162.820, Y  +443.809, Z    +0.000, E1   -22.804, E3 +604058.955}
SPL {X  -162.820, Y  +447.077, Z    +0.000, E1   -22.869, E3 +604074.765}
SPL {X  -162.820, Y  +449.911, Z    +0.000, E1   -22.774, E3 +604089.375}
SPL {X  -162.820, Y  +451.861, Z    +0.000, E1   -22.750, E3 +604099.222}
SPL {X  -162.820, Y  +454.167, Z    +0.000, E1   -22.842, E3 +604109.952}
SPL {X  -162.820, Y  +456.529, Z    +0.000, E1   -22.855, E3 +604121.480}
SPL {X  -162.820, Y  +458.725, Z    +0.000, E1   -22.793, E3 +604132.885}
SPL {X  -162.820, Y  +461.700, Z    +0.000, E1   -22.822, E3 +604147.507}
SPL {X  -162.820, Y  +464.633, Z    +0.000, E1   -22.813, E3 +604162.004}
SPL {X  -162.820, Y  +466.699, Z    +0.000, E1   -22.824, E3 +604172.050}
SPL {X  -162.820, Y  +468.655, Z    +0.000, E1   -22.858, E3 +604181.494}
SPL {X  -162.820, Y  +470.892, Z    +0.000, E1   -22.837, E3 +604192.732}
SPL {X  -162.820, Y  +473.485, Z    +0.000, E1   -22.806, E3 +604205.931}
SPL {X  -162.820, Y  +475.738, Z    +0.000, E1   -22.728, E3 +604217.596}
SPL {X  -162.820, Y  +478.177, Z    +0.000, E1   -22.834, E3 +604228.935}
SPL {X  -162.820, Y  +481.034, Z    +0.000, E1   -22.831, E3 +604243.073}
SPL {X  -162.820, Y  +483.391, Z    +0.000, E1   -22.793, E3 +604255.009}
SPL {X  -162.820, Y  +486.307, Z    +0.000, E1   -22.833, E3 +604269.263}
SPL {X  -162.820, Y  +489.750, Z    +0.000, E1   -22.832, E3 +604286.333}
SPL {X  -162.820, Y  +492.546, Z    +0.000, E1   -22.823, E3 +604300.091}
SPL {X  -162.820, Y  +495.526, Z    +0.000, E1   -22.833, E3 +604314.974}
SPL {X  -162.820, Y  +499.330, Z    +0.000, E1   -22.841, E3 +604333.755}
SPL {X  -162.820, Y  +502.361, Z    +0.000, E1   -22.801, E3 +604348.913}
SPL {X  -162.820, Y  +505.323, Z    +0.000, E1   -22.838, E3 +604363.385}
SPL {X  -162.820, Y  +508.611, Z    +0.000, E1   -22.838, E3 +604379.648}
SPL {X  -162.820, Y  +511.620, Z    +0.000, E1   -22.791, E3 +604394.892}
SPL {X  -162.820, Y  +513.873, Z    +0.000, E1   -22.800, E3 +604405.864}
SPL {X  -162.820, Y  +516.100, Z    +0.000, E1   -22.809, E3 +604416.940}
SPL {X  -162.820, Y  +518.662, Z    +0.000, E1   -22.847, E3 +604429.239}
SPL {X  -162.820, Y  +520.641, Z    +0.000, E1   -22.790, E3 +604439.480}
SPL {X  -162.820, Y  +522.740, Z    +0.000, E1   -22.811, E3 +604449.723}
SPL {X  -162.820, Y  +524.628, Z    +0.000, E1   -22.846, E3 +604458.718}
SPL {X  -162.820, Y  +526.661, Z    +0.000, E1   -22.801, E3 +604469.273}
SPL {X  -162.820, Y  +529.662, Z    +0.000, E1   -22.810, E3 +604484.124}
SPL {X  -162.820, Y  +532.614, Z    +0.000, E1   -22.828, E3 +604498.530}
SPL {X  -162.820, Y  +534.838, Z    +0.000, E1   -22.864, E3 +604509.159}
SPL {X  -162.820, Y  +536.882, Z    +0.000, E1   -22.782, E3 +604520.014}
SPL {X  -162.820, Y  +539.194, Z    +0.000, E1   -22.826, E3 +604531.062}
SPL {X  -162.820, Y  +541.555, Z    +0.000, E1   -22.817, E3 +604542.877}
SPL {X  -162.820, Y  +543.728, Z    +0.000, E1   -22.799, E3 +604553.734}
SPL {X  -162.820, Y  +545.925, Z    +0.000, E1   -22.803, E3 +604564.604}
SPL {X  -162.820, Y  +548.328, Z    +0.000, E1   -22.796, E3 +604576.600}
SPL {X  -162.820, Y  +551.027, Z    +0.000, E1   -22.819, E3 +604589.792}
SPL {X  -162.820, Y  +553.721, Z    +0.000, E1   -22.807, E3 +604603.237}
SPL {X  -162.820, Y  +556.430, Z    +0.000, E1   -22.821, E3 +604616.532}
SPL {X  -162.820, Y  +559.675, Z    +0.000, E1   -22.837, E3 +604632.613}
SPL {X  -162.820, Y  +562.799, Z    +0.000, E1   -22.814, E3 +604648.119}
SPL {X  -162.820, Y  +565.170, Z    +0.000, E1   -22.801, E3 +604659.944}
SPL {X  -162.820, Y  +568.020, Z    +0.000, E1   -22.787, E3 +604674.330}
SPL {X  -162.820, Y  +570.992, Z    +0.000, E1   -22.834, E3 +604688.550}
SPL {X  -162.820, Y  +572.901, Z    +0.000, E1   -22.775, E3 +604698.418}
SPL {X  -162.820, Y  +575.638, Z    +0.000, E1   -22.855, E3 +604711.528}
SPL {X  -162.820, Y  +578.553, Z    +0.000, E1   -22.801, E3 +604726.240}
SPL {X  -162.820, Y  +581.064, Z    +0.000, E1   -22.823, E3 +604738.524}
SPL {X  -162.820, Y  +583.435, Z    +0.000, E1   -22.808, E3 +604750.346}
SPL {X  -162.820, Y  +585.410, Z    +0.000, E1   -22.764, E3 +604760.482}
SPL {X  -162.820, Y  +587.676, Z    +0.000, E1   -22.853, E3 +604770.996}
SPL {X  -162.820, Y  +589.682, Z    +0.000, E1   -22.776, E3 +604781.526}
SPL {X  -162.820, Y  +591.720, Z    +0.000, E1   -22.868, E3 +604790.837}
SPL {X  -162.820, Y  +593.650, Z    +0.000, E1   -22.810, E3 +604800.907}
SPL {X  -162.820, Y  +595.830, Z    +0.000, E1   -22.828, E3 +604811.523}
SPL {X  -162.820, Y  +598.094, Z    +0.000, E1   -22.843, E3 +604822.636}
SPL {X  -162.820, Y  +600.420, Z    +0.000, E1   -22.826, E3 +604834.267}
SPL {X  -162.820, Y  +602.573, Z    +0.000, E1   -22.830, E3 +604844.852}
SPL {X  -162.820, Y  +604.828, Z    +0.000, E1   -22.784, E3 +604856.491}
SPL {X  -162.820, Y  +607.142, Z    +0.000, E1   -22.808, E3 +604867.671}
SPL {X  -162.820, Y  +608.890, Z    +0.000, E1   -22.790, E3 +604876.496}
SPL {X  -162.820, Y  +611.103, Z    +0.000, E1   -22.785, E3 +604887.534}
SPL {X  -162.820, Y  +613.294, Z    +0.000, E1   -22.780, E3 +604898.407}
SPL {X  -162.820, Y  +615.356, Z    +0.000, E1   -22.799, E3 +604908.464}
SPL {X  -162.820, Y  +617.439, Z    +0.000, E1   -22.808, E3 +604918.723}
SPL {X  -162.820, Y  +619.665, Z    +0.000, E1   -22.817, E3 +604929.691}
SPL {X  -162.820, Y  +621.733, Z    +0.000, E1   -22.759, E3 +604940.415}
SPL {X  -162.820, Y  +624.076, Z    +0.000, E1   -22.774, E3 +604951.920}
SPL {X  -162.820, Y  +626.527, Z    +0.000, E1   -22.768, E3 +604964.162}
SPL {X  -162.820, Y  +629.758, Z    +0.000, E1   -22.800, E3 +604980.091}
SPL {X  -162.820, Y  +632.572, Z    +0.000, E1   -22.785, E3 +604993.941}
SPL {X  -162.820, Y  +634.507, Z    +0.000, E1   -22.784, E3 +605003.579}
SPL {X  -162.820, Y  +636.863, Z    +0.000, E1   -22.760, E3 +605015.502}
SPL {X  -162.820, Y  +640.111, Z    +0.000, E1   -22.809, E3 +605031.384}
SPL {X  -162.820, Y  +643.449, Z    +0.000, E1   -22.796, E3 +605047.902}
SPL {X  -162.820, Y  +645.630, Z    +0.000, E1   -22.795, E3 +605058.598}
SPL {X  -162.820, Y  +647.561, Z    +0.000, E1   -22.705, E3 +605069.049}
SPL {X  -162.820, Y  +649.758, Z    +0.000, E1   -22.780, E3 +605079.239}
SPL {X  -162.820, Y  +651.708, Z    +0.000, E1   -22.810, E3 +605088.733}
SPL {X  -162.820, Y  +653.898, Z    +0.000, E1   -22.796, E3 +605099.654}
SPL {X  -162.820, Y  +656.161, Z    +0.000, E1   -22.812, E3 +605110.776}
SPL {X  -162.820, Y  +658.384, Z    +0.000, E1   -22.822, E3 +605121.642}
SPL {X  -162.820, Y  +660.215, Z    +0.000, E1   -22.649, E3 +605132.233}
SPL {X  -162.820, Y  +662.823, Z    +0.000, E1   -22.799, E3 +605143.941}
SPL {X  -162.820, Y  +665.112, Z    +0.000, E1   -22.835, E3 +605154.995}
SPL {X  -162.820, Y  +667.016, Z    +0.000, E1   -22.823, E3 +605164.423}
SPL {X  -162.820, Y  +668.960, Z    +0.000, E1   -22.773, E3 +605174.591}
SPL {X  -162.820, Y  +672.333, Z    +0.000, E1   -22.837, E3 +605190.927}
SPL {X  -162.812, Y  +675.071, Z    +0.000, E1   -22.742, E3 +605205.072}
SPL {X  -162.773, Y  +677.428, Z    +0.000, E1   -22.762, E3 +605216.669}
SPL {X  -162.691, Y  +679.987, Z    +0.000, E1   -22.794, E3 +605229.083}
SPL {X  -162.604, Y  +681.880, Z    +0.000, E1   -22.691, E3 +605239.244}
SPL {X  -162.458, Y  +684.346, Z    +0.000, E1   -22.764, E3 +605251.037}
SPL {X  -162.296, Y  +686.547, Z    +0.000, E1   -22.660, E3 +605262.654}
SPL {X  -162.090, Y  +688.902, Z    +0.000, E1   -22.700, E3 +605274.162}
SPL {X  -161.474, Y  +694.390, Z    +0.000, E1   -24.298, E3 +605287.517}
SPL {X  -158.730, Y  +709.763, Z    +0.000, E1   -31.225, E3 +605298.856}
ENDSPLINE

SPLINE
SPL {X  -160.932, Y  +698.225, Z    +0.000, E1   -21.712, E3 +605329.965}
SPL {X  -161.917, Y  +690.622, Z    +0.000, E1   -16.445, E3 +605343.566}
ENDSPLINE

SPLINE
SPL {X  -161.349, Y  +695.340, Z    +0.000, E1   -18.625, E3 +605351.185}
ENDSPLINE

SPLINE
SPL {X  -162.534, Y  +683.153, Z    +0.000, E1   -10.475, E3 +605372.315}
SPL {X  -162.820, Y  +667.630, Z    +0.000, E1    -0.882, E3 +605366.292}
SPL {X  -162.820, Y  +661.883, Z    +0.000, E1    +3.373, E3 +605371.735}
SPL {X  -162.820, Y  +653.808, Z    +0.000, E1    +9.891, E3 +605369.426}
SPL {X  -162.820, Y  +632.548, Z    +0.000, E1   +27.446, E3 +605365.963}
ENDSPLINE

SPLINE
SPL {X  -162.820, Y  +638.080, Z    +0.000, E1   +18.858, E3 +605393.711}
ENDSPLINE

SPLINE
SPL {X  -162.820, Y  +623.278, Z    +0.000, E1   +28.723, E3 +605395.282}
SPL {X  -162.820, Y  +618.658, Z    +0.000, E1   +26.841, E3 +605423.891}
ENDSPLINE

SPLINE
SPL {X  -162.820, Y  +623.685, Z    +0.000, E1   +22.346, E3 +605436.197}
ENDSPLINE

SPLINE
SPL {X  -162.820, Y  +621.304, Z    +0.000, E1   +22.259, E3 +605449.013}
SPL {X  -162.820, Y  +618.758, Z    +0.000, E1   +22.239, E3 +605462.163}
SPL {X  -162.820, Y  +616.062, Z    +0.000, E1   +22.275, E3 +605475.584}
SPL {X  -162.820, Y  +613.536, Z    +0.000, E1   +22.242, E3 +605488.706}
SPL {X  -162.820, Y  +610.461, Z    +0.000, E1   +22.264, E3 +605504.337}
SPL {X  -162.820, Y  +606.755, Z    +0.000, E1   +22.275, E3 +605523.135}
SPL {X  -162.820, Y  +603.020, Z    +0.000, E1   +22.272, E3 +605542.195}
SPL {X  -162.820, Y  +599.168, Z    +0.000, E1   +22.310, E3 +605561.463}
SPL {X  -162.820, Y  +595.597, Z    +0.000, E1   +22.284, E3 +605579.799}
SPL {X  -162.820, Y  +592.389, Z    +0.000, E1   +22.245, E3 +605596.402}
SPL {X  -162.820, Y  +589.492, Z    +0.000, E1   +22.304, E3 +605610.586}
SPL {X  -162.820, Y  +587.447, Z    +0.000, E1   +22.279, E3 +605621.115}
SPL {X  -162.820, Y  +585.192, Z    +0.000, E1   +22.298, E3 +605632.525}
SPL {X  -162.820, Y  +582.610, Z    +0.000, E1   +22.234, E3 +605646.149}
SPL {X  -162.820, Y  +580.317, Z    +0.000, E1   +22.300, E3 +605657.203}
SPL {X  -162.820, Y  +578.878, Z    +0.000, E1   +22.272, E3 +605664.712}
SPL {X  -162.820, Y  +576.856, Z    +0.000, E1   +22.233, E3 +605675.471}
SPL {X  -162.820, Y  +574.811, Z    +0.000, E1   +22.236, E3 +605685.734}
SPL {X  -162.820, Y  +572.645, Z    +0.000, E1   +22.246, E3 +605696.830}
SPL {X  -162.820, Y  +569.475, Z    +0.000, E1   +22.269, E3 +605712.836}
SPL {X  -162.820, Y  +565.838, Z    +0.000, E1   +22.271, E3 +605731.431}
SPL {X  -162.820, Y  +562.162, Z    +0.000, E1   +22.252, E3 +605750.248}
SPL {X  -162.820, Y  +558.919, Z    +0.000, E1   +22.286, E3 +605766.411}
SPL {X  -162.820, Y  +556.169, Z    +0.000, E1   +22.295, E3 +605780.240}
SPL {X  -162.820, Y  +553.294, Z    +0.000, E1   +22.266, E3 +605795.238}
SPL {X  -162.820, Y  +550.136, Z    +0.000, E1   +22.258, E3 +605811.351}
SPL {X  -162.820, Y  +546.694, Z    +0.000, E1   +22.290, E3 +605828.673}
SPL {X  -162.820, Y  +543.558, Z    +0.000, E1   +22.285, E3 +605844.536}
SPL {X  -162.820, Y  +541.633, Z    +0.000, E1   +22.257, E3 +605854.464}
SPL {X  -162.820, Y  +539.116, Z    +0.000, E1   +22.302, E3 +605867.075}
SPL {X  -162.820, Y  +535.523, Z    +0.000, E1   +22.266, E3 +605885.737}
SPL {X  -162.820, Y  +531.757, Z    +0.000, E1   +22.276, E3 +605904.791}
SPL {X  -162.820, Y  +527.980, Z    +0.000, E1   +22.326, E3 +605923.622}
SPL {X  -162.820, Y  +524.599, Z    +0.000, E1   +22.287, E3 +605941.020}
SPL {X  -162.820, Y  +522.011, Z    +0.000, E1   +22.282, E3 +605954.096}
SPL {X  -162.820, Y  +519.457, Z    +0.000, E1   +22.481, E3 +605965.386}
SPL {X  -162.820, Y  +505.859, Z    +0.000, E1   +28.367, E3 +605979.869}
SPL {X  -162.820, Y  +504.131, Z    +0.000, E1   +27.325, E3 +605994.007}
SPL {X  -162.820, Y  +503.215, Z    +0.000, E1   +26.369, E3 +606004.693}
SPL {X  -162.820, Y  +502.265, Z    +0.000, E1   +25.287, E3 +606017.175}
SPL {X  -162.820, Y  +501.060, Z    +0.000, E1   +24.081, E3 +606031.916}
SPL {X  -162.820, Y  +500.336, Z    +0.000, E1   +23.110, E3 +606043.056}
SPL {X  -162.820, Y  +499.247, Z    +0.000, E1   +22.302, E3 +606055.457}
ENDSPLINE

SLIN {X  -200.000, Y  +530.000, E1    +0.000}
HALT
END
